(* IEC 61131-3 sources: ArfBotOS/Codesys-4/ArfBotOS.fbsdev/Application.iecapp^/FUN, 8 files *)

(* ---- F_AddElement.fn.st ---- *)
FUNCTION F_AddElement
VAR_IN_OUT
	Command: STRING(GVL_App.COMMAND_LEN);
END_VAR
VAR_INPUT
	Delimiter: STRING(1):=' '; // default to space
	Element: STRING(GVL_App.COMMAND_LEN);
END_VAR
VAR
END_VAR

//
// input
// 	Element: 'bar'
// 	Delimiter: ','
// 	Command: 'foo'
//
// output
// 	Command: 'foo,bar'
//

Command:=CONCAT(Command, Element);
Command:=CONCAT(Command, Delimiter);
END_FUNCTION

(* ---- F_AxisErrorDetail.fn.st ---- *)
FUNCTION F_AxisErrorDetail : STRING(255)
VAR_IN_OUT
	Axis: AXIS_REF_SM3;
END_VAR
VAR_INPUT
	AxisName: STRING(8);
END_VAR
VAR
	_i: INT;
	_id: SMC_ERROR;
	_s: STRING(255);
	_root: STRING(180);
	_stop: STRING(180);
	_inst: STRING(80);
END_VAR

(* Decode the SoftMotion FB that actually put this axis in errorstop.
   AXIS_REF.fbeFBError[].wID is the real SMC_ERROR (following error, SW limit, ...).
   Code 183 (SMC_MS_AXIS_IN_ERRORSTOP) is only "Stop cannot be executed" after
   the axis is already faulted -- skip it when a root cause is present. *)
F_AxisErrorDetail := '';
IF (NOT Axis.bError) AND (Axis.nAxisState <> SMC_AXIS_STATE.errorstop) THEN
	RETURN;
END_IF

_s := AxisName;
_root := '';
_stop := '';

FOR _i := 0 TO g_SMC_NUMBER_FB_ERRORS DO
	_id := Axis.fbeFBError[_i].wID;
	IF _id <> SMC_NO_ERROR THEN
		_inst := Axis.fbeFBError[_i].strErrorInstance;
		IF (_id = SMC_MS_AXIS_IN_ERRORSTOP) OR (_id = SMC_H_AXIS_IN_ERRORSTOP) THEN
			IF _stop = '' THEN
				_stop := CONCAT(TO_STRING(_id), CONCAT(' ', SMC_ErrorString(_id, SMC_Language_Type.english)));
			END_IF
		ELSIF _root = '' THEN
			_root := CONCAT(TO_STRING(_id), CONCAT(' ', SMC_ErrorString(_id, SMC_Language_Type.english)));
			IF _inst <> '' THEN
				_root := CONCAT(_root, CONCAT(' [', CONCAT(_inst, ']')));
			END_IF
		END_IF
	END_IF
END_FOR

IF _root <> '' THEN
	_s := CONCAT(_s, CONCAT(' ', _root));
ELSIF _stop <> '' THEN
	_s := CONCAT(_s, CONCAT(' ', _stop));
ELSE
	_s := CONCAT(_s, ' errorstop');
END_IF

IF Axis.dwErrorID <> 0 THEN
	_s := CONCAT(_s, CONCAT(' drive ', DWORD_TO_STRING(Axis.dwErrorID)));
END_IF

F_AxisErrorDetail := _s;
END_FUNCTION

(* ---- F_Checksum.fn.st ---- *)
FUNCTION F_Checksum : UINT
VAR_INPUT
	data: POINTER TO BYTE;
	length: UINT;
END_VAR
VAR
	curr_crc: UINT;
	sum1, sum2: USINT;
	_i, _j, _k: UINT;
END_VAR

// https://www.tutorialspoint.com/cyclic-redundancy-check-crc-in-arduino
curr_crc := 16#0000;
sum1 := UINT_TO_USINT(curr_crc);
sum2 := UINT_TO_USINT(SHR(curr_crc, 8));
FOR _i:=0 TO length - 1 BY 1 DO
	sum1 := (sum1 + data[_i]) MOD 255;
	sum2 := (sum2 + sum1) MOD 255;
END_FOR
{warning disable C0308}
F_Checksum := SHL(sum2, 8) OR sum1;
{warning restore C0308}
END_FUNCTION

(* ---- F_RadToDeg.fn.st ---- *)
FUNCTION F_RadToDeg : LREAL
VAR_INPUT
    Radians: LREAL;
END_VAR
VAR
END_VAR

F_RadToDeg := Radians * (180 / GVL_App.pi);
END_FUNCTION

(* ---- F_RoundLreal.fn.st ---- *)
FUNCTION F_RoundLreal : LREAL
VAR_INPUT
   rIn : LREAL;
   Digit: INT;
END_VAR

VAR
   d1 : DINT;
   r0,r1,r2,Rdigit: LREAL;
END_VAR

// https://forge.codesys.com/forge/talk/Engineering/thread/8d1ee86294/
rdigit   :=INT_TO_LREAL(Digit);
r0 := EXPT(10,rdigit);
r1 := rIn * r0;
d1 := TRUNC(r1);
r2 := DINT_TO_LREAL(d1);
F_RoundLreal := r2 / r0;
END_FUNCTION

(* ---- F_RoundToInt.fn.st ---- *)
(* Round LREAL to nearest INT (half away from zero via ±0.5 then truncate).
   LREAL_TO_INT alone truncates toward zero (27.8->27, -27.8->-27), which
   systematically under-drives |Hz| and biases crawl toward stop.
   Positive: add 0.5 then LREAL_TO_INT. Negative: subtract 0.5 then LREAL_TO_INT
   so both sides round to nearest (e.g. 27.8->28, -27.8->-28).
   Used when converting LREAL step rate (Hz) to INT16 for the Teensy PTO. *)

FUNCTION F_RoundToInt : INT
VAR_INPUT
	x : LREAL;
END_VAR
VAR
END_VAR

IF x >= 0.0 THEN
    F_RoundToInt := LREAL_TO_INT(x + 0.5);
ELSE
    F_RoundToInt := LREAL_TO_INT(x - 0.5);
END_IF
END_FUNCTION

(* ---- FB_CommandProcessor.fb.st ---- *)
FUNCTION_BLOCK FB_CommandProcessor EXTENDS FB_Module
VAR_IN_OUT
	J1, J2, J3, J4, J5, J6: AXIS_REF_SM3;
	AxisGroup: AXIS_GROUP_REF_SM3;
	GroupHandler: FB_GroupHandler;
	CmdIO: ST_LogicCmdIO;
	PrgProcessor: FB_ProgramProcessor;
END_VAR
VAR_INPUT
	Enable: BOOL;
END_VAR
VAR_OUTPUT
	ItfActiveProcessorUnitMode: PACK_ML.IUnitMode;
	ItfActiveModule: ItfModule;
	StatusText: STRING(255);
    GCodeLines: ARRAY[0..SMC_GCodeViewer.c_uiLines] OF STRING;
END_VAR
VAR
	_Commands: ARRAY [GVL_App.PROG_CMDS_ARR_BEG..GVL_App.PROG_CMDS_ARR_END] OF DUT_Command;
	_DummyUnitMode: PACK_ML.UnitMode;
	_UnitModeCurrentState: PACK_ML.State;
	_ActiveCommand: DUT_Command;
	_CurrentCmdIdx: UINT;
	_ProcessMoveCommand: FB_MoveCmdProcessor;
	_ProcessPauseCommand: FB_PauseCmdProcessor;
	//_ProcessInputCommand: InputCommandProcessor;
	_ProcessOutputCommand: FB_OutputCmdProcessor;
	_ProcessorDoneRtrig: R_TRIG;
    _ProcessVisionCommand: REFERENCE TO FB_VisionCmdProcessor; // keep vision in separate task
	_ProcessVarSetCommand: FB_VarSetCmdProcessor;
	_ProcessCncCommand: FB_CncCmdProcessor;
	_ProcessLogicCommand: FB_LogicCmdProcessor;
    _ErrorRtrig: ARRAY[0..7] OF R_TRIG;
	_FirstScan: BOOL:=TRUE;
END_VAR

VAR CONSTANT
	_STEP_DONE: 			INT := 1000;
	_STEP_IDLE: 			INT := 0000;
	_STEP_CMD:				INT := 0010;
	_STEP_WAIT:				INT := 0020;
	_STEP_ERR:              INT := 0030;
END_VAR

// keep this reference at the top in case we reference this somewhere else first
// hint: originally this was an issue because of the done and reset bits being referenced first
_ProcessVisionCommand REF= _40_Vision.ProcessVisionCommand;

//
SUPER^();

//
IF _FirstScan THEN
	// will exception if we don't set this on first scan
	_DummyUnitMode(sName := 'Active Processor',
					eInitialState := PACK_ML.State.Idle,
					xActive := TRUE);
	ItfActiveProcessorUnitMode := _DummyUnitMode;
END_IF

// this is at best a hack and needs to be rethought out.
// we logically cant assign a process as the active unit mode
// at start up so we use this dummy one
CASE _DummyUnitMode.CurrentState OF
	PACK_ML.State.Stopped,
	PACK_ML.State.Aborted,
	PACK_ML.State.Held,
	PACK_ML.State.Suspended,
	PACK_ML.State.Complete,
	PACK_ML.State.Idle:
		//
	PACK_ML.State.Resetting,
	PACK_ML.State.Starting,
	PACK_ML.State.Execute,
	PACK_ML.State.Suspending,
	PACK_ML.State.UnSuspending,
	PACK_ML.State.Holding,
	PACK_ML.State.UnHolding,
	PACK_ML.State.Completing,
	PACK_ML.State.Aborting,
	PACK_ML.State.Stopping,
	PACK_ML.State.Clearing:
		_DummyUnitMode.ActingStateCompleted();
END_CASE

// PackML state machine implementation
_UnitModeCurrentState := SUPER^._UnitMode.CurrentState;

//
_ErrorRtrig[0](CLK:=_ProcessMoveCommand.Error);
IF _ErrorRtrig[0].Q THEN
	SUPER^.M_Error(Description:=CONCAT('Move Error: ', _ProcessMoveCommand.ErrorDescription));
	StatusText:=SUPER^.ErrorDescription;
END_IF
_ErrorRtrig[1](CLK:=_ProcessPauseCommand.Error);
IF _ErrorRtrig[1].Q THEN
	SUPER^.M_Error(Description:=CONCAT('Pause Error: ', _ProcessPauseCommand.ErrorDescription));
	StatusText:=SUPER^.ErrorDescription;
END_IF
(*
_ErrorRtrig[2](CLK:=_ProcessInputCommand.Error);
IF _ErrorRtrig[2].Q THEN
	SUPER^._M_Error(Description:=CONCAT('Input Error: ', _ProcessInputCommand.ErrorDescription));
	StatusText:=SUPER^.ErrorDescription;
END_IF*)
_ErrorRtrig[3](CLK:=_ProcessOutputCommand.Error);
IF _ErrorRtrig[3].Q THEN
	SUPER^.M_Error(Description:=CONCAT('Output Error: ', _ProcessOutputCommand.ErrorDescription));
	StatusText:=SUPER^.ErrorDescription;
END_IF
_ErrorRtrig[4](CLK:=_ProcessVisionCommand.Error);
IF _ErrorRtrig[4].Q THEN
	SUPER^.M_Error(Description:=CONCAT('Vision Error: ', _ProcessVisionCommand.ErrorDescription));
	StatusText:=SUPER^.ErrorDescription;
END_IF
_ErrorRtrig[5](CLK:=_ProcessVarSetCommand.Error);
IF _ErrorRtrig[5].Q THEN
	SUPER^.M_Error(Description:=CONCAT('Variable Error: ', _ProcessVarSetCommand.ErrorDescription));
	StatusText:=SUPER^.ErrorDescription;
END_IF
_ErrorRtrig[6](CLK:=_ProcessCncCommand.Error);
IF _ErrorRtrig[6].Q THEN
	SUPER^.M_Error(Description:=CONCAT('CNC Error: ', _ProcessCncCommand.ErrorDescription));
	StatusText:=SUPER^.ErrorDescription;
END_IF
_ErrorRtrig[7](CLK:=_ProcessLogicCommand.Error);
IF _ErrorRtrig[7].Q THEN
	SUPER^.M_Error(Description:=CONCAT('Logic Error: ', _ProcessLogicCommand.ErrorDescription));
	StatusText:=SUPER^.ErrorDescription;
END_IF

_ProcessMoveCommand(
	StoredPositions:= SUPER^.StoredPositions,
	VisionRegisters:= SUPER^.VisionRegisters,
	Flags:= SUPER^.Flags,
	AxisGroup:= AxisGroup,
	GroupHandler:= GroupHandler,
	Velocity:= PersistentVars.StoredPositions[GVL_App.SPEEDS_IDX].Position.X,
	VelFactor:= PersistentVars.StoredPositions[GVL_App.SPEEDS_IDX].Position.A,
	Acceleration:= PersistentVars.StoredPositions[GVL_App.SPEEDS_IDX].Position.Y,
	AccFactor:= PersistentVars.StoredPositions[GVL_App.SPEEDS_IDX].Position.B,
	Jerk:= PersistentVars.StoredPositions[GVL_App.SPEEDS_IDX].Position.Z,
	JerkFactor:= PersistentVars.StoredPositions[GVL_App.SPEEDS_IDX].Position.C,
	Position=> ,
	ItfUnitMode=>,
	Error=> );

_ProcessPauseCommand(
	StoredPositions:= SUPER^.StoredPositions,
	VisionRegisters:= SUPER^.VisionRegisters,
	Flags:= SUPER^.Flags,
	ElapsedTime=> ,
	RemainingTime=> ,
	ItfUnitMode=>,
	Error=> );

//_ProcessInputCommand();
_ProcessOutputCommand(
	StoredPositions:= SUPER^.StoredPositions,
	VisionRegisters:= SUPER^.VisionRegisters,
	Flags:= SUPER^.Flags,
	Digital:= CmdIO.Output,
	Pwm:= CmdIO.Pwm,
	Enable:= Enable,
	ItfUnitMode=>,
	Error=> );

_ProcessVarSetCommand(
	StoredPositions:= SUPER^.StoredPositions,
	VisionRegisters:= SUPER^.VisionRegisters,
	Flags:= SUPER^.Flags,
	ItfUnitMode=>,
	Error=> ,
	ErrorDescription=> );

_ProcessCncCommand(
	StoredPositions:= SUPER^.StoredPositions,
	VisionRegisters:= SUPER^.VisionRegisters,
	Flags:= SUPER^.Flags,
	J1:=J1, J2:=J2, J3:=J3, J4:=J4, J5:=J5, J6:=J6,
	AxisGroup:= AxisGroup,
    CmdIO:= CmdIO,
    GCodeLines => GCodeLines,
	GapJerk:= ,
	GapVelocity:= ,
	AvoidGaps:= ,
	GapAccel:= ,
	ItfUnitMode=>,
	Error=> ,
	ErrorDescription=> );

_ProcessLogicCommand(
	StoredPositions:= SUPER^.StoredPositions,
	VisionRegisters:= SUPER^.VisionRegisters,
	Flags:= SUPER^.Flags,
	CmdProcessor:= THIS^,
	PrgProcessor:= PrgProcessor,
	ItfUnitMode=>,
	Error=> ,
	ErrorDescription=> ,
	CmdIO:= CmdIO);

_FirstScan := FALSE;
END_FUNCTION_BLOCK

(* ---- FB_ProgramProcessor.fb.st ---- *)
FUNCTION_BLOCK FB_ProgramProcessor EXTENDS FB_Module
VAR_IN_OUT
	Programs: ARRAY [GVL_App.PROG_ARR_BEG..GVL_App.PROG_ARR_END] OF DUT_Program;
	J1, J2, J3, J4, J5, J6: AXIS_REF_SM3;
	AxisGroup: AXIS_GROUP_REF_SM3;
	GroupHandler: FB_GroupHandler;
	CmdIO: ST_LogicCmdIO;
END_VAR
VAR_INPUT
	Enable: BOOL;
END_VAR
VAR_OUTPUT
	ItfActiveProcessorUnitMode	: PACK_ML.IUnitMode;
	ItfActiveModule: ItfModule;
	StatusText: STRING(255);
    GCodeLines: ARRAY[0..SMC_GCodeViewer.c_uiLines] OF STRING;
END_VAR
VAR
	_DummyUnitMode: PACK_ML.UnitMode;
	_UnitModeCurrentState: PACK_ML.State;
	_Returning:  ARRAY [GVL_App.PROG_ARR_BEG..GVL_App.PROG_ARR_END] OF BOOL;
	_ReturnPrograms: ARRAY [GVL_App.PROG_ARR_BEG..GVL_App.PROG_ARR_END] OF UINT;
	_ReturnCommands: ARRAY [GVL_App.PROG_CMDS_ARR_BEG..GVL_App.PROG_CMDS_ARR_END + 1] OF UINT; // +1 because we want to be able to tell if calling program was on last command
	_CurrentPrgIdx: UINT;
	_ProcessCommands: FB_CommandProcessor;
	_Commands: ARRAY [GVL_App.PROG_CMDS_ARR_BEG..GVL_App.PROG_CMDS_ARR_END] OF DUT_Command;
    _ErrorRtrig: R_TRIG;
	_i, _j, _k: INT;
	_FirstScan: BOOL:=TRUE;
END_VAR

VAR CONSTANT
	_STEP_DONE: 			INT := 1000;
	_STEP_IDLE: 			INT := 0000;
	_STEP_PRG:				INT := 0010;
	_STEP_WAIT_EXECUTE:		INT := 0020;
	_STEP_WAIT_IDLE:		INT := 0025;
	_STEP_ERR:              INT := 0030;
END_VAR

//
SUPER^();

//
IF _FirstScan THEN
	// will exception if we don't set this on first scan
	_DummyUnitMode(sName := 'Active Processor',
					eInitialState := PACK_ML.State.Idle,
					xActive := TRUE);
	ItfActiveProcessorUnitMode := _DummyUnitMode;
END_IF

// this is at best a hack and needs to be rethought out.
// we logically cant assign a process as the active unit mode
// at start up so we use this dummy one
CASE _DummyUnitMode.CurrentState OF
	PACK_ML.State.Stopped,
	PACK_ML.State.Aborted,
	PACK_ML.State.Held,
	PACK_ML.State.Suspended,
	PACK_ML.State.Complete,
	PACK_ML.State.Idle:
		//
	PACK_ML.State.Resetting,
	PACK_ML.State.Starting,
	PACK_ML.State.Execute,
	PACK_ML.State.Suspending,
	PACK_ML.State.UnSuspending,
	PACK_ML.State.Holding,
	PACK_ML.State.UnHolding,
	PACK_ML.State.Completing,
	PACK_ML.State.Aborting,
	PACK_ML.State.Stopping,
	PACK_ML.State.Clearing:
		_DummyUnitMode.ActingStateCompleted();
END_CASE

// PackML state machine implementation
_UnitModeCurrentState := SUPER^._UnitMode.CurrentState;

//
_ErrorRtrig(CLK:=_ProcessCommands.Error);
IF _ErrorRtrig.Q THEN
	SUPER^.M_Error(Description:=CONCAT('Command Processor Error: ', _ProcessCommands.ErrorDescription));
	StatusText:=SUPER^.ErrorDescription;
END_IF

//
_ProcessCommands(
	StoredPositions:=SUPER^.StoredPositions,
	VisionRegisters:=SUPER^.VisionRegisters,
	Flags:=SUPER^.Flags,
	J1:=J1, J2:=J2, J3:=J3, J4:=J4, J5:=J5, J6:=J6,
	AxisGroup:= AxisGroup,
	GroupHandler:= GroupHandler,
	CmdIO:=CmdIO,
	PrgProcessor:= THIS^,
    GCodeLines => GCodeLines,
	Enable:= Enable,
	Error=> ,
	StatusText=>StatusText);

_FirstScan := FALSE;
END_FUNCTION_BLOCK
